(* Logix 5000 project; controller LeakTestAuto vendor 1 type 14 code 226 rev 37.11; software revision 37.01; part 10 of 13 *)
(* tags used below, declared in another part *)
   AOI_Barcode_Comms : AOI_CommStatus;
   AOI_CTS1 : AOI_CTS_INSTRUMENT;
   AOI_CTS1_Comms : AOI_CommStatus;
   AOI_CTS2 : AOI_CTS_INSTRUMENT;
   AOI_CTS2_Comms : AOI_CommStatus;
   AOI_RFID_Comms : AOI_CommStatus;
   AOI_Robot_Comms : AOI_CommStatus;
   AOI_SeqSteps : AOI_StandardSeqSteps;
   BarcodeScanner : udt_OutputStructure;
   Conveyor : udt_OutputStructure;
   Conveyor_Seq : udt_SequenceStructure_X64;
   ConveyorCleatSensorFault : BOOL;
   CTS1_Seq : udt_SequenceStructure_X64;
   CTS2_Seq : udt_SequenceStructure_X64;
   FailCount : COUNTER;
   LastFaults : DINT[2];
   LeakTester1 : udt_OutputStructure;
   LeakTester2 : udt_OutputStructure;
   Nest1Bypass : BOOL;
   Nest1Cylinder : udt_OutputStructure;
   Nest2Bypass : BOOL;
   Nest2Cylinder : udt_OutputStructure;
   ONS_ClearWarnings : BOOL;
   OP220 : udt_Mode;
   OP220_Fault_Counter : COUNTER;
   OP220_Fault_Counter_ONS : BOOL;
   OP220_Fault_Number : DINT;
   OP220_Fault_Reset_ONS : BOOL;
   OP220_FaultCounter_Reset_ONS : BOOL;
   OP220_HomingSeq : udt_SequenceStructure_X64;
   OP220_LeakTest : udt_ProcessFault;
   OP220_Seq : udt_SequenceStructure_X64;
   RFID_Cylinder1_Mismatch : BOOL;
   RFID_Cylinder2_Mismatch : BOOL;
   RFIDScanner : udt_OutputStructure;
   Robot : udt_OutputStructure;
   RobotGripper : udt_OutputStructure;
   TON_Cylinder1DownTimeout : TIMER;
   TON_Cylinder1UpTimeout : TIMER;
   TON_Cylinder2DownTimeout : TIMER;
   TON_Cylinder2UpTimeout : TIMER;
   TON_FailChute : TIMER[10];
   I_OP220_N3_REJECT_BIN_OK : ALIAS FOR Local:3:I.Pt09.Data;
   I_OP220_N4_DC_OK : ALIAS FOR Local:4:I.Pt01.Data;
   I_OP220_N4_DC_OK_PS2 : ALIAS FOR Local:4:I.Pt04.Data;
   OP220_ConsumedFromMain_RobotPickupSafe : BOOL;
   OP220_EStopTest_DCS : DCI_STOP;
   PLC : AOI_PLC;
   ShiftChange : BOOL;
(* MainProgram, continued *)

ROUTINE R90_Faults   (* ladder *)
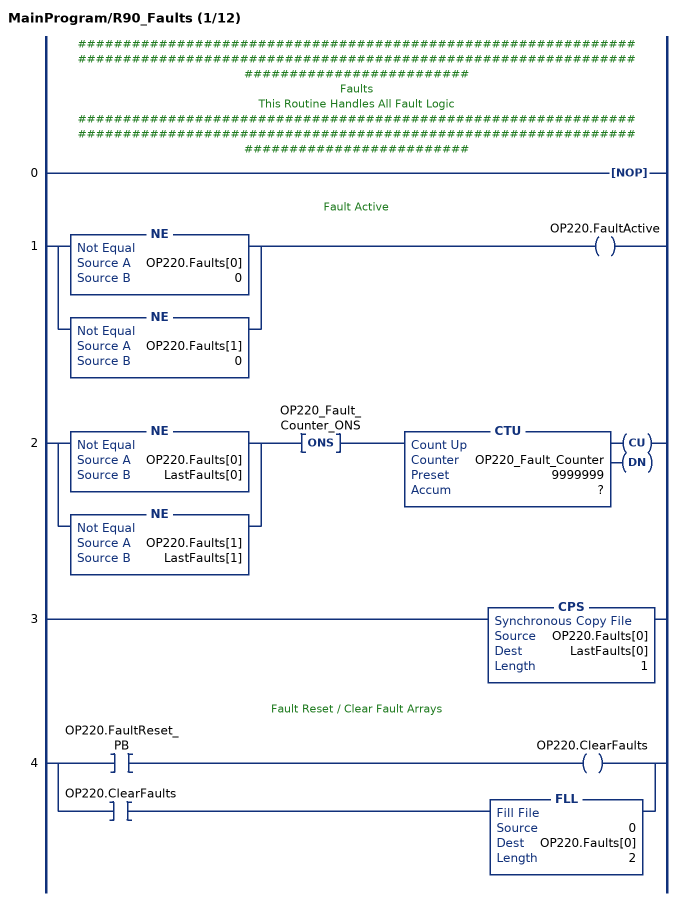
   // #####################################################################################################################################################
   // Faults
   // This Routine Handles All Fault Logic
   // #####################################################################################################################################################
   0: NOP();
   // Fault Active
   1: [NE(OP220.Faults[0],0) ,NE(OP220.Faults[1],0) ]OTE(OP220.FaultActive);
   2: [NE(OP220.Faults[0],LastFaults[0]) ,NE(OP220.Faults[1],LastFaults[1]) ]ONS(OP220_Fault_Counter_ONS)CTU(OP220_Fault_Counter,?,?);
   3: CPS(OP220.Faults[0],LastFaults[0],1);
   // Fault Reset / Clear Fault Arrays
   4: [XIC(OP220.FaultReset_PB) OTE(OP220.ClearFaults) ,XIC(OP220.ClearFaults) FLL(0,OP220.Faults[0],2) ];
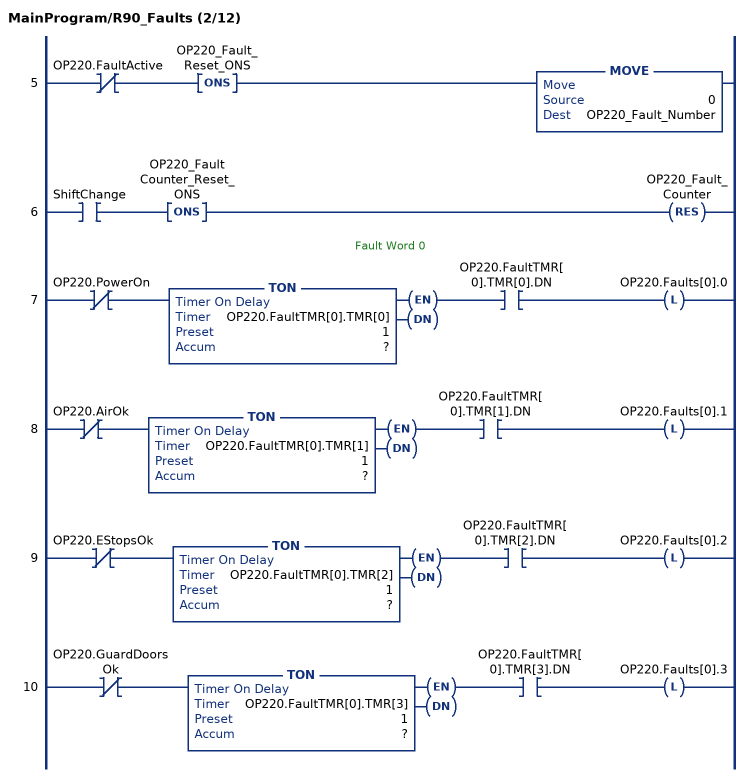
   5: XIO(OP220.FaultActive)ONS(OP220_Fault_Reset_ONS)MOVE(0,OP220_Fault_Number);
   6: XIC(ShiftChange)ONS(OP220_FaultCounter_Reset_ONS)RES(OP220_Fault_Counter);
   // Fault Word 0
   7: XIO(OP220.PowerOn)TON(OP220.FaultTMR[0].TMR[0],?,?)XIC(OP220.FaultTMR[0].TMR[0].DN)OTL(OP220.Faults[0].0);
   8: XIO(OP220.AirOk)TON(OP220.FaultTMR[0].TMR[1],?,?)XIC(OP220.FaultTMR[0].TMR[1].DN)OTL(OP220.Faults[0].1);
   9: XIO(OP220.EStopsOk)TON(OP220.FaultTMR[0].TMR[2],?,?)XIC(OP220.FaultTMR[0].TMR[2].DN)OTL(OP220.Faults[0].2);
   10: XIO(OP220.GuardDoorsOk)TON(OP220.FaultTMR[0].TMR[3],?,?)XIC(OP220.FaultTMR[0].TMR[3].DN)OTL(OP220.Faults[0].3);
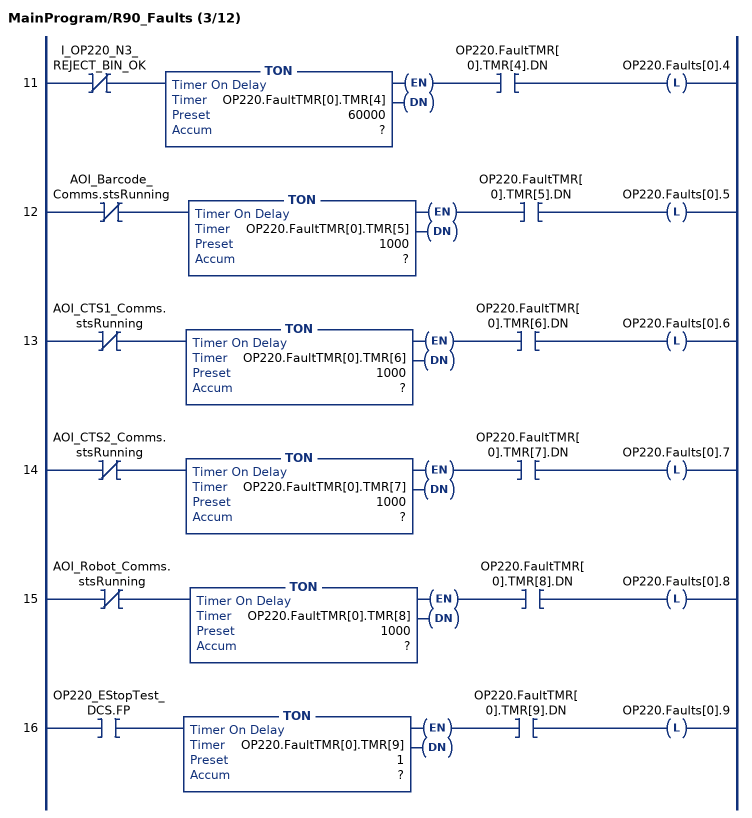
   11: XIO(I_OP220_N3_REJECT_BIN_OK)TON(OP220.FaultTMR[0].TMR[4],?,?)XIC(OP220.FaultTMR[0].TMR[4].DN)OTL(OP220.Faults[0].4);
   12: XIO(AOI_Barcode_Comms.stsRunning)TON(OP220.FaultTMR[0].TMR[5],?,?)XIC(OP220.FaultTMR[0].TMR[5].DN)OTL(OP220.Faults[0].5);
   13: XIO(AOI_CTS1_Comms.stsRunning)TON(OP220.FaultTMR[0].TMR[6],?,?)XIC(OP220.FaultTMR[0].TMR[6].DN)OTL(OP220.Faults[0].6);
   14: XIO(AOI_CTS2_Comms.stsRunning)TON(OP220.FaultTMR[0].TMR[7],?,?)XIC(OP220.FaultTMR[0].TMR[7].DN)OTL(OP220.Faults[0].7);
   15: XIO(AOI_Robot_Comms.stsRunning)TON(OP220.FaultTMR[0].TMR[8],?,?)XIC(OP220.FaultTMR[0].TMR[8].DN)OTL(OP220.Faults[0].8);
   16: XIC(OP220_EStopTest_DCS.FP)TON(OP220.FaultTMR[0].TMR[9],?,?)XIC(OP220.FaultTMR[0].TMR[9].DN)OTL(OP220.Faults[0].9);
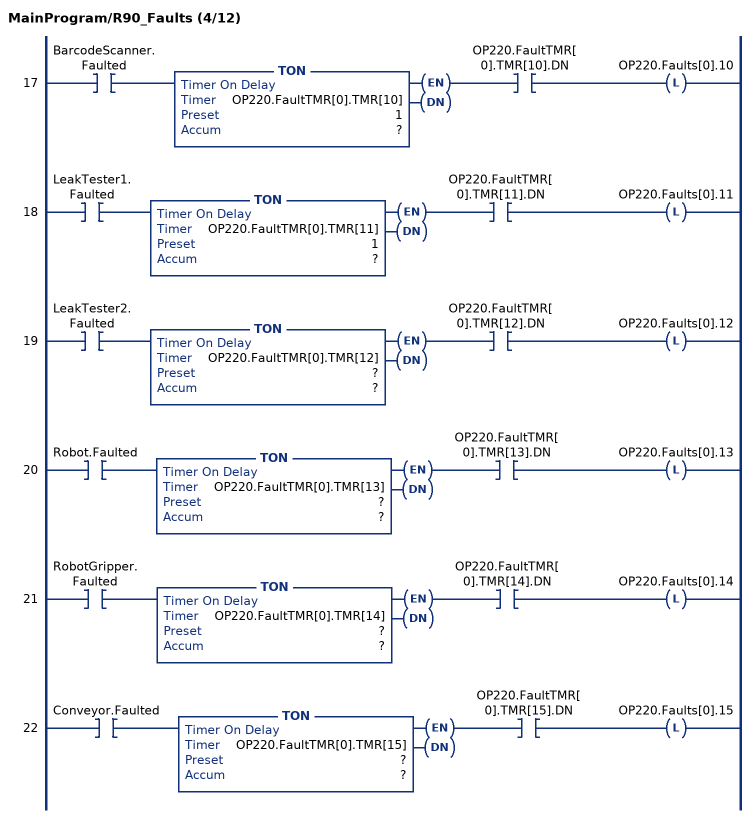
   17: XIC(BarcodeScanner.Faulted)TON(OP220.FaultTMR[0].TMR[10],?,?)XIC(OP220.FaultTMR[0].TMR[10].DN)OTL(OP220.Faults[0].10);
   18: XIC(LeakTester1.Faulted)TON(OP220.FaultTMR[0].TMR[11],?,?)XIC(OP220.FaultTMR[0].TMR[11].DN)OTL(OP220.Faults[0].11);
   19: XIC(LeakTester2.Faulted)TON(OP220.FaultTMR[0].TMR[12],?,?)XIC(OP220.FaultTMR[0].TMR[12].DN)OTL(OP220.Faults[0].12);
   20: XIC(Robot.Faulted)TON(OP220.FaultTMR[0].TMR[13],?,?)XIC(OP220.FaultTMR[0].TMR[13].DN)OTL(OP220.Faults[0].13);
   21: XIC(RobotGripper.Faulted)TON(OP220.FaultTMR[0].TMR[14],?,?)XIC(OP220.FaultTMR[0].TMR[14].DN)OTL(OP220.Faults[0].14);
   22: XIC(Conveyor.Faulted)TON(OP220.FaultTMR[0].TMR[15],?,?)XIC(OP220.FaultTMR[0].TMR[15].DN)OTL(OP220.Faults[0].15);
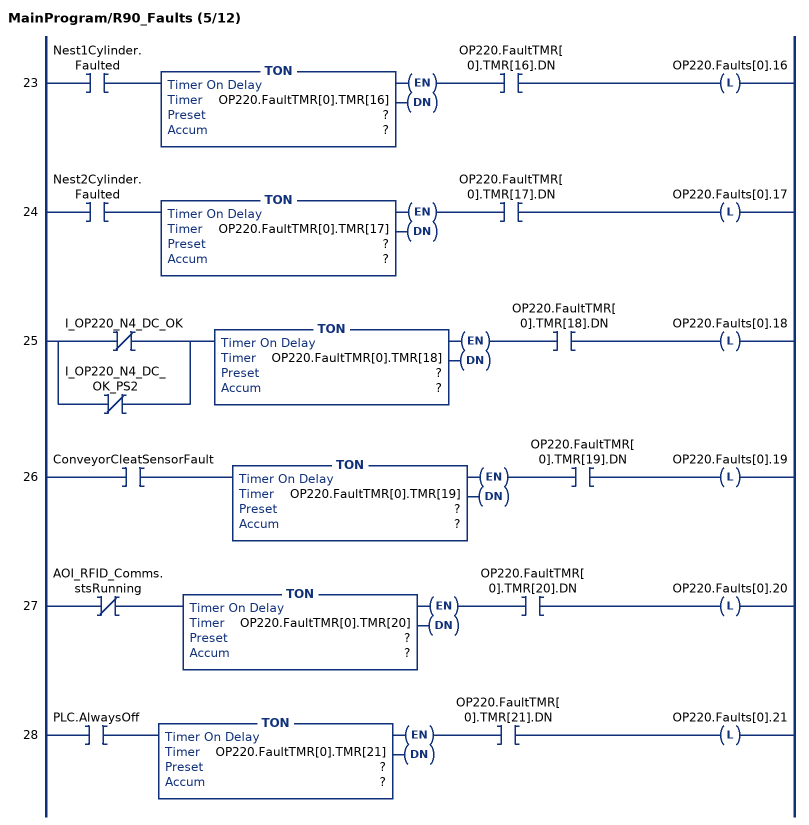
   23: XIC(Nest1Cylinder.Faulted)TON(OP220.FaultTMR[0].TMR[16],?,?)XIC(OP220.FaultTMR[0].TMR[16].DN)OTL(OP220.Faults[0].16);
   24: XIC(Nest2Cylinder.Faulted)TON(OP220.FaultTMR[0].TMR[17],?,?)XIC(OP220.FaultTMR[0].TMR[17].DN)OTL(OP220.Faults[0].17);
   25: [XIO(I_OP220_N4_DC_OK) ,XIO(I_OP220_N4_DC_OK_PS2) ]TON(OP220.FaultTMR[0].TMR[18],?,?)XIC(OP220.FaultTMR[0].TMR[18].DN)OTL(OP220.Faults[0].18);
   26: XIC(ConveyorCleatSensorFault)TON(OP220.FaultTMR[0].TMR[19],?,?)XIC(OP220.FaultTMR[0].TMR[19].DN)OTL(OP220.Faults[0].19);
   27: XIO(AOI_RFID_Comms.stsRunning)TON(OP220.FaultTMR[0].TMR[20],?,?)XIC(OP220.FaultTMR[0].TMR[20].DN)OTL(OP220.Faults[0].20);
   28: XIC(PLC.AlwaysOff)TON(OP220.FaultTMR[0].TMR[21],?,?)XIC(OP220.FaultTMR[0].TMR[21].DN)OTL(OP220.Faults[0].21);
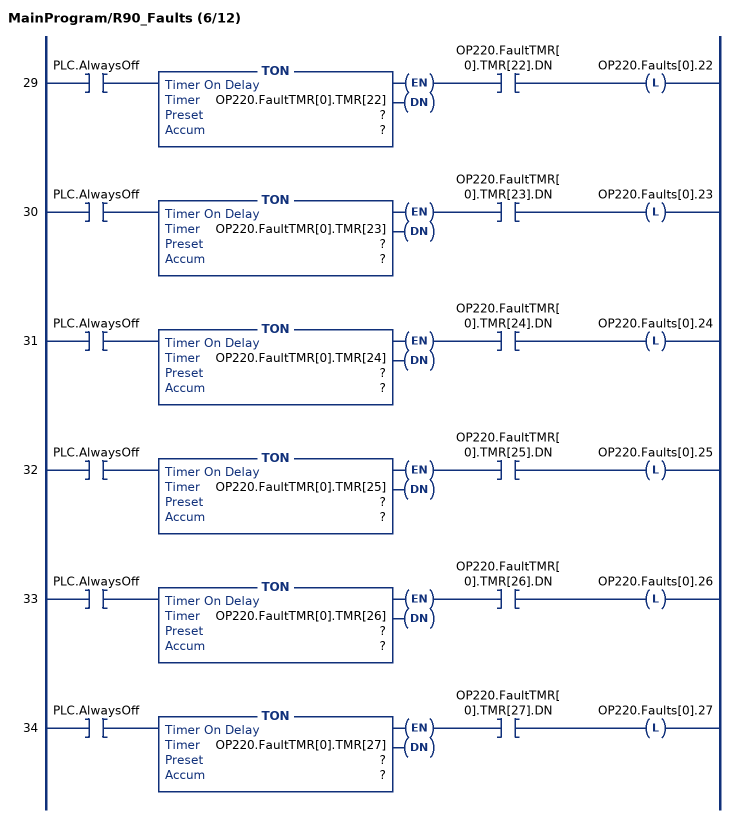
   29: XIC(PLC.AlwaysOff)TON(OP220.FaultTMR[0].TMR[22],?,?)XIC(OP220.FaultTMR[0].TMR[22].DN)OTL(OP220.Faults[0].22);
   30: XIC(PLC.AlwaysOff)TON(OP220.FaultTMR[0].TMR[23],?,?)XIC(OP220.FaultTMR[0].TMR[23].DN)OTL(OP220.Faults[0].23);
   31: XIC(PLC.AlwaysOff)TON(OP220.FaultTMR[0].TMR[24],?,?)XIC(OP220.FaultTMR[0].TMR[24].DN)OTL(OP220.Faults[0].24);
   32: XIC(PLC.AlwaysOff)TON(OP220.FaultTMR[0].TMR[25],?,?)XIC(OP220.FaultTMR[0].TMR[25].DN)OTL(OP220.Faults[0].25);
   33: XIC(PLC.AlwaysOff)TON(OP220.FaultTMR[0].TMR[26],?,?)XIC(OP220.FaultTMR[0].TMR[26].DN)OTL(OP220.Faults[0].26);
   34: XIC(PLC.AlwaysOff)TON(OP220.FaultTMR[0].TMR[27],?,?)XIC(OP220.FaultTMR[0].TMR[27].DN)OTL(OP220.Faults[0].27);
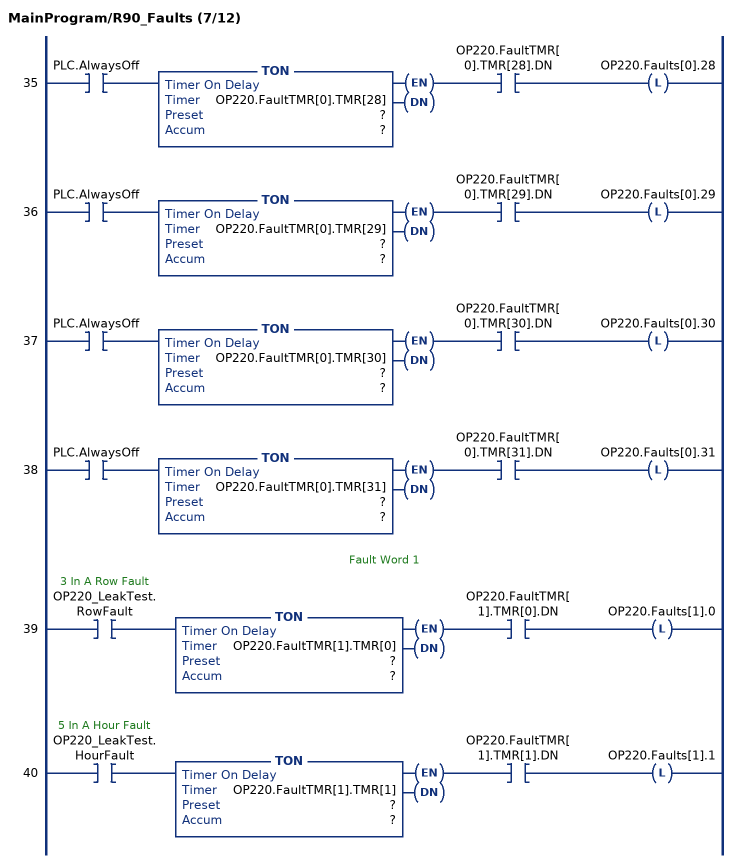
   35: XIC(PLC.AlwaysOff)TON(OP220.FaultTMR[0].TMR[28],?,?)XIC(OP220.FaultTMR[0].TMR[28].DN)OTL(OP220.Faults[0].28);
   36: XIC(PLC.AlwaysOff)TON(OP220.FaultTMR[0].TMR[29],?,?)XIC(OP220.FaultTMR[0].TMR[29].DN)OTL(OP220.Faults[0].29);
   37: XIC(PLC.AlwaysOff)TON(OP220.FaultTMR[0].TMR[30],?,?)XIC(OP220.FaultTMR[0].TMR[30].DN)OTL(OP220.Faults[0].30);
   38: XIC(PLC.AlwaysOff)TON(OP220.FaultTMR[0].TMR[31],?,?)XIC(OP220.FaultTMR[0].TMR[31].DN)OTL(OP220.Faults[0].31);
   // Fault Word 1
   39: XIC(OP220_LeakTest.RowFault)TON(OP220.FaultTMR[1].TMR[0],?,?)XIC(OP220.FaultTMR[1].TMR[0].DN)OTL(OP220.Faults[1].0);
   40: XIC(OP220_LeakTest.HourFault)TON(OP220.FaultTMR[1].TMR[1],?,?)XIC(OP220.FaultTMR[1].TMR[1].DN)OTL(OP220.Faults[1].1);
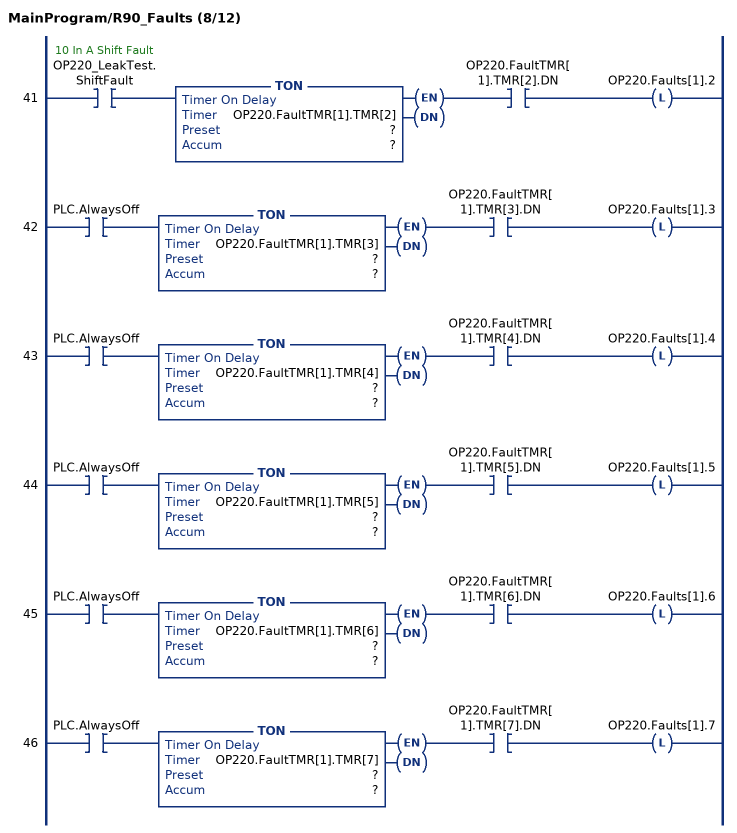
   41: XIC(OP220_LeakTest.ShiftFault)TON(OP220.FaultTMR[1].TMR[2],?,?)XIC(OP220.FaultTMR[1].TMR[2].DN)OTL(OP220.Faults[1].2);
   42: XIC(PLC.AlwaysOff)TON(OP220.FaultTMR[1].TMR[3],?,?)XIC(OP220.FaultTMR[1].TMR[3].DN)OTL(OP220.Faults[1].3);
   43: XIC(PLC.AlwaysOff)TON(OP220.FaultTMR[1].TMR[4],?,?)XIC(OP220.FaultTMR[1].TMR[4].DN)OTL(OP220.Faults[1].4);
   44: XIC(PLC.AlwaysOff)TON(OP220.FaultTMR[1].TMR[5],?,?)XIC(OP220.FaultTMR[1].TMR[5].DN)OTL(OP220.Faults[1].5);
   45: XIC(PLC.AlwaysOff)TON(OP220.FaultTMR[1].TMR[6],?,?)XIC(OP220.FaultTMR[1].TMR[6].DN)OTL(OP220.Faults[1].6);
   46: XIC(PLC.AlwaysOff)TON(OP220.FaultTMR[1].TMR[7],?,?)XIC(OP220.FaultTMR[1].TMR[7].DN)OTL(OP220.Faults[1].7);
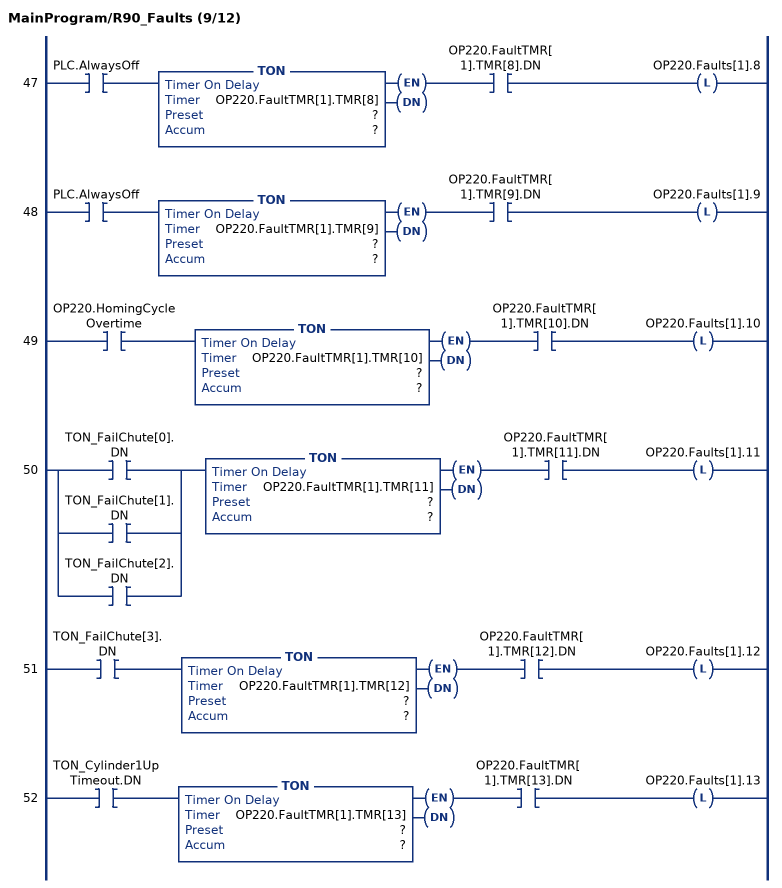
   47: XIC(PLC.AlwaysOff)TON(OP220.FaultTMR[1].TMR[8],?,?)XIC(OP220.FaultTMR[1].TMR[8].DN)OTL(OP220.Faults[1].8);
   48: XIC(PLC.AlwaysOff)TON(OP220.FaultTMR[1].TMR[9],?,?)XIC(OP220.FaultTMR[1].TMR[9].DN)OTL(OP220.Faults[1].9);
   49: XIC(OP220.HomingCycleOvertime)TON(OP220.FaultTMR[1].TMR[10],?,?)XIC(OP220.FaultTMR[1].TMR[10].DN)OTL(OP220.Faults[1].10);
   50: [XIC(TON_FailChute[0].DN) ,XIC(TON_FailChute[1].DN) ,XIC(TON_FailChute[2].DN) ]TON(OP220.FaultTMR[1].TMR[11],?,?)XIC(OP220.FaultTMR[1].TMR[11].DN)OTL(OP220.Faults[1].11);
   51: XIC(TON_FailChute[3].DN)TON(OP220.FaultTMR[1].TMR[12],?,?)XIC(OP220.FaultTMR[1].TMR[12].DN)OTL(OP220.Faults[1].12);
   52: XIC(TON_Cylinder1UpTimeout.DN)TON(OP220.FaultTMR[1].TMR[13],?,?)XIC(OP220.FaultTMR[1].TMR[13].DN)OTL(OP220.Faults[1].13);
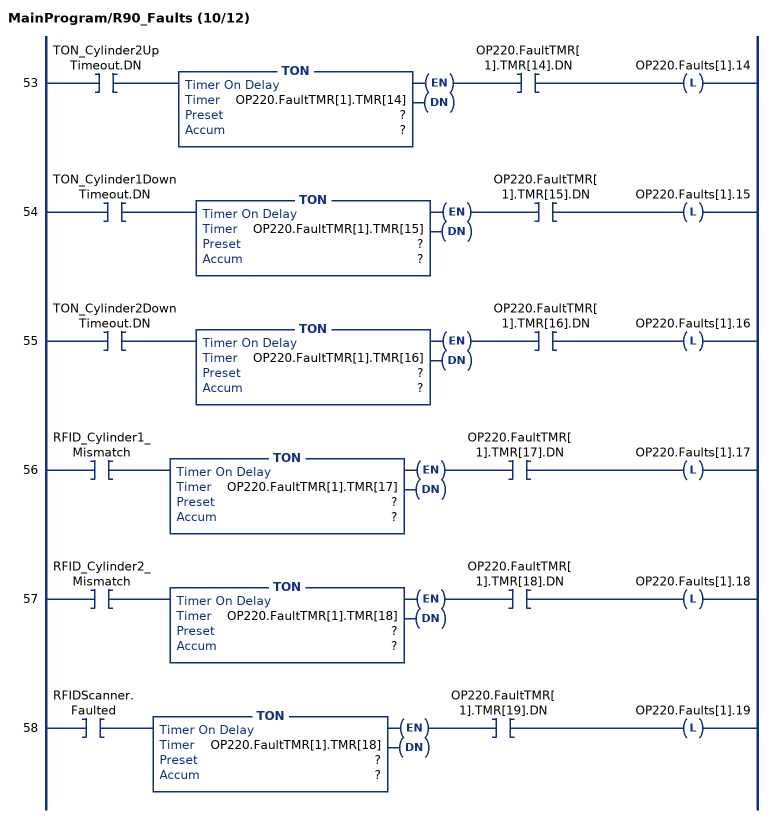
   53: XIC(TON_Cylinder2UpTimeout.DN)TON(OP220.FaultTMR[1].TMR[14],?,?)XIC(OP220.FaultTMR[1].TMR[14].DN)OTL(OP220.Faults[1].14);
   54: XIC(TON_Cylinder1DownTimeout.DN)TON(OP220.FaultTMR[1].TMR[15],?,?)XIC(OP220.FaultTMR[1].TMR[15].DN)OTL(OP220.Faults[1].15);
   55: XIC(TON_Cylinder2DownTimeout.DN)TON(OP220.FaultTMR[1].TMR[16],?,?)XIC(OP220.FaultTMR[1].TMR[16].DN)OTL(OP220.Faults[1].16);
   56: XIC(RFID_Cylinder1_Mismatch)TON(OP220.FaultTMR[1].TMR[17],?,?)XIC(OP220.FaultTMR[1].TMR[17].DN)OTL(OP220.Faults[1].17);
   57: XIC(RFID_Cylinder2_Mismatch)TON(OP220.FaultTMR[1].TMR[18],?,?)XIC(OP220.FaultTMR[1].TMR[18].DN)OTL(OP220.Faults[1].18);
   58: XIC(RFIDScanner.Faulted)TON(OP220.FaultTMR[1].TMR[18],?,?)XIC(OP220.FaultTMR[1].TMR[19].DN)OTL(OP220.Faults[1].19);
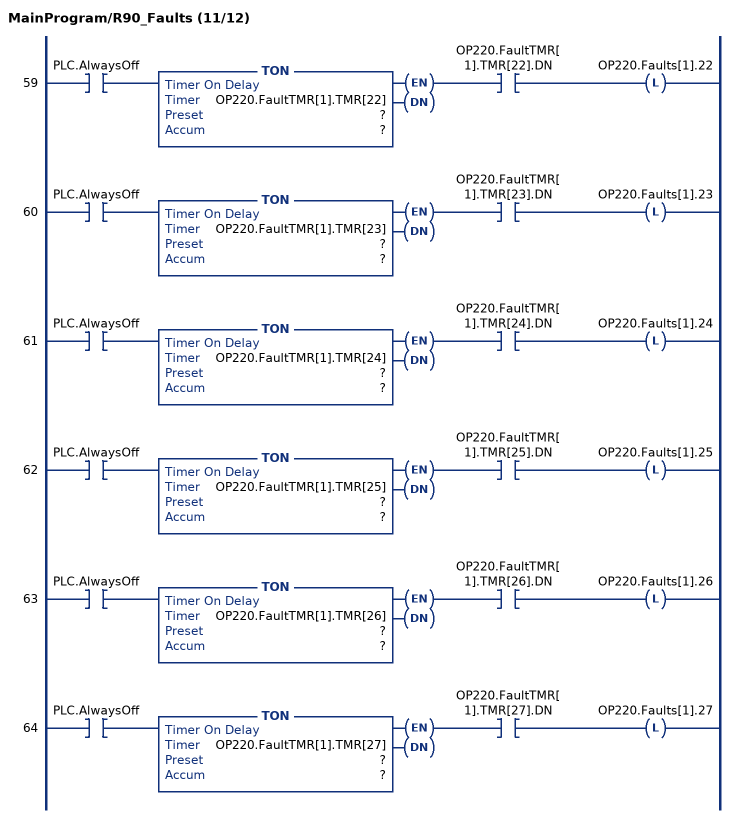
   59: XIC(PLC.AlwaysOff)TON(OP220.FaultTMR[1].TMR[22],?,?)XIC(OP220.FaultTMR[1].TMR[22].DN)OTL(OP220.Faults[1].22);
   60: XIC(PLC.AlwaysOff)TON(OP220.FaultTMR[1].TMR[23],?,?)XIC(OP220.FaultTMR[1].TMR[23].DN)OTL(OP220.Faults[1].23);
   61: XIC(PLC.AlwaysOff)TON(OP220.FaultTMR[1].TMR[24],?,?)XIC(OP220.FaultTMR[1].TMR[24].DN)OTL(OP220.Faults[1].24);
   62: XIC(PLC.AlwaysOff)TON(OP220.FaultTMR[1].TMR[25],?,?)XIC(OP220.FaultTMR[1].TMR[25].DN)OTL(OP220.Faults[1].25);
   63: XIC(PLC.AlwaysOff)TON(OP220.FaultTMR[1].TMR[26],?,?)XIC(OP220.FaultTMR[1].TMR[26].DN)OTL(OP220.Faults[1].26);
   64: XIC(PLC.AlwaysOff)TON(OP220.FaultTMR[1].TMR[27],?,?)XIC(OP220.FaultTMR[1].TMR[27].DN)OTL(OP220.Faults[1].27);
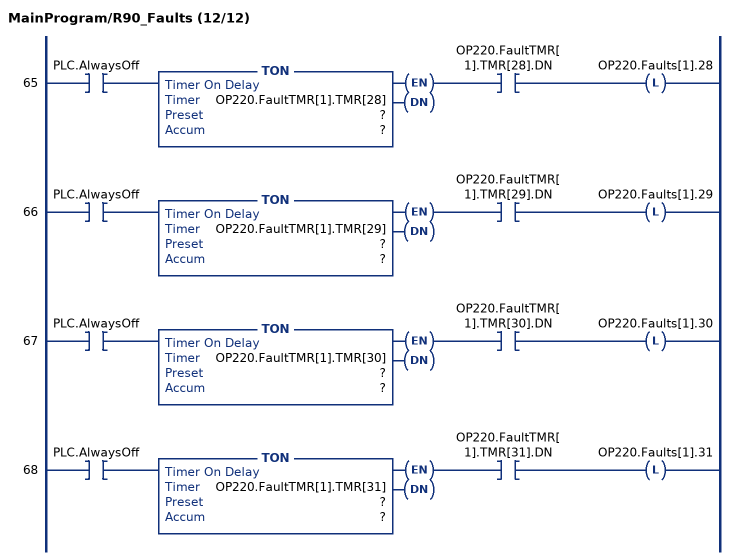
   65: XIC(PLC.AlwaysOff)TON(OP220.FaultTMR[1].TMR[28],?,?)XIC(OP220.FaultTMR[1].TMR[28].DN)OTL(OP220.Faults[1].28);
   66: XIC(PLC.AlwaysOff)TON(OP220.FaultTMR[1].TMR[29],?,?)XIC(OP220.FaultTMR[1].TMR[29].DN)OTL(OP220.Faults[1].29);
   67: XIC(PLC.AlwaysOff)TON(OP220.FaultTMR[1].TMR[30],?,?)XIC(OP220.FaultTMR[1].TMR[30].DN)OTL(OP220.Faults[1].30);
   68: XIC(PLC.AlwaysOff)TON(OP220.FaultTMR[1].TMR[31],?,?)XIC(OP220.FaultTMR[1].TMR[31].DN)OTL(OP220.Faults[1].31);
END_ROUTINE

ROUTINE R91_Warnings   (* ladder *)
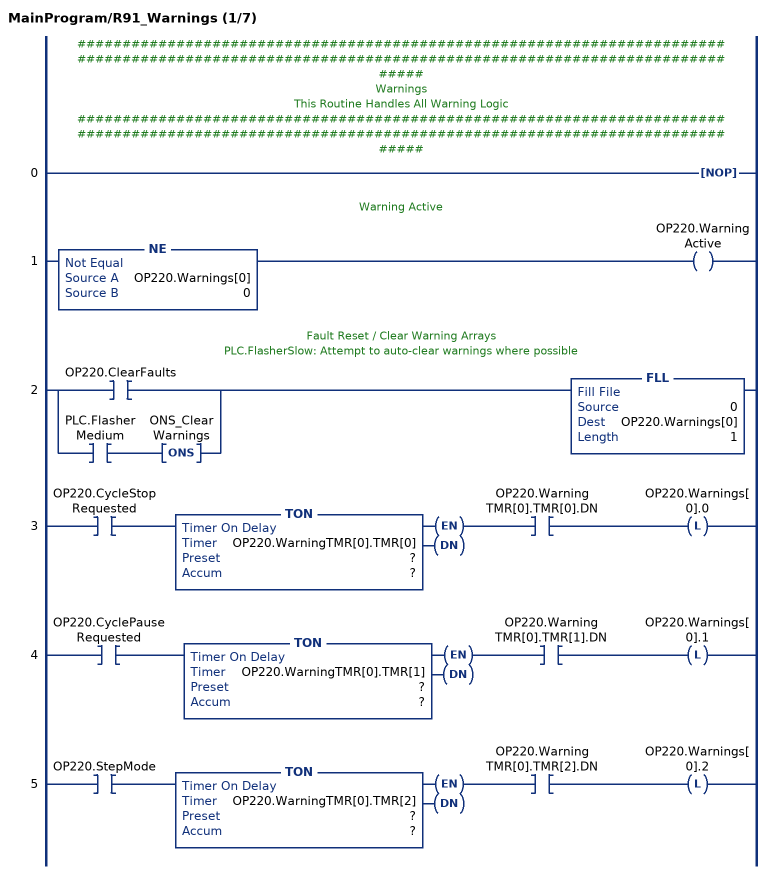
   // #####################################################################################################################################################
   // Warnings
   // This Routine Handles All Warning Logic
   // #####################################################################################################################################################
   0: NOP();
   // Warning Active
   1: NE(OP220.Warnings[0],0)OTE(OP220.WarningActive);
   // Fault Reset / Clear Warning Arrays
   // PLC.FlasherSlow: Attempt to auto-clear warnings where possible
   2: [XIC(OP220.ClearFaults) ,XIC(PLC.FlasherMedium) ONS(ONS_ClearWarnings) ]FLL(0,OP220.Warnings[0],1);
   3: XIC(OP220.CycleStopRequested)TON(OP220.WarningTMR[0].TMR[0],?,?)XIC(OP220.WarningTMR[0].TMR[0].DN)OTL(OP220.Warnings[0].0);
   4: XIC(OP220.CyclePauseRequested)TON(OP220.WarningTMR[0].TMR[1],?,?)XIC(OP220.WarningTMR[0].TMR[1].DN)OTL(OP220.Warnings[0].1);
   5: XIC(OP220.StepMode)TON(OP220.WarningTMR[0].TMR[2],?,?)XIC(OP220.WarningTMR[0].TMR[2].DN)OTL(OP220.Warnings[0].2);
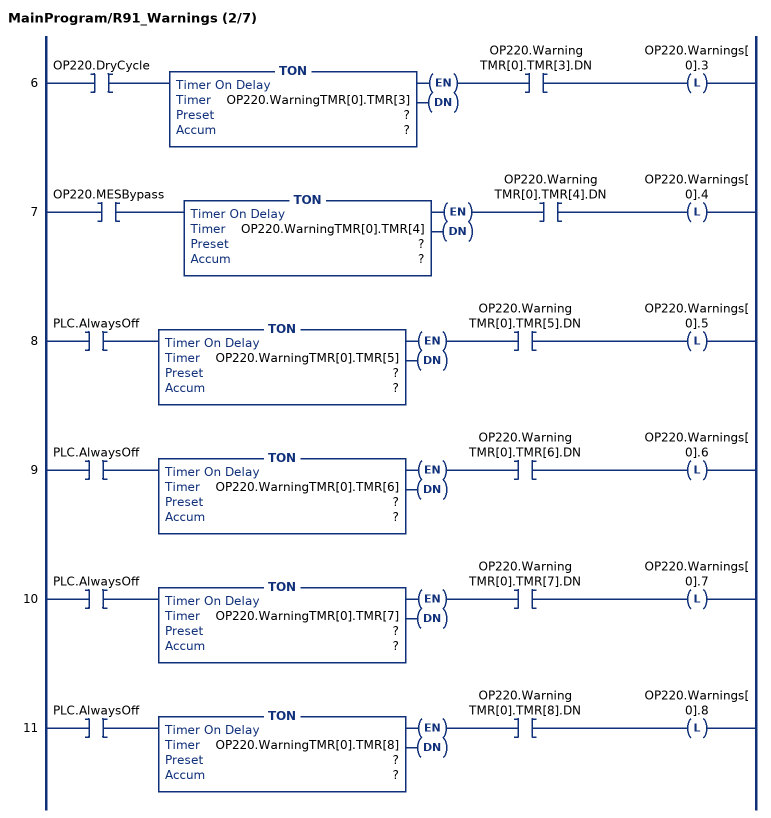
   6: XIC(OP220.DryCycle)TON(OP220.WarningTMR[0].TMR[3],?,?)XIC(OP220.WarningTMR[0].TMR[3].DN)OTL(OP220.Warnings[0].3);
   7: XIC(OP220.MESBypass)TON(OP220.WarningTMR[0].TMR[4],?,?)XIC(OP220.WarningTMR[0].TMR[4].DN)OTL(OP220.Warnings[0].4);
   8: XIC(PLC.AlwaysOff)TON(OP220.WarningTMR[0].TMR[5],?,?)XIC(OP220.WarningTMR[0].TMR[5].DN)OTL(OP220.Warnings[0].5);
   9: XIC(PLC.AlwaysOff)TON(OP220.WarningTMR[0].TMR[6],?,?)XIC(OP220.WarningTMR[0].TMR[6].DN)OTL(OP220.Warnings[0].6);
   10: XIC(PLC.AlwaysOff)TON(OP220.WarningTMR[0].TMR[7],?,?)XIC(OP220.WarningTMR[0].TMR[7].DN)OTL(OP220.Warnings[0].7);
   11: XIC(PLC.AlwaysOff)TON(OP220.WarningTMR[0].TMR[8],?,?)XIC(OP220.WarningTMR[0].TMR[8].DN)OTL(OP220.Warnings[0].8);
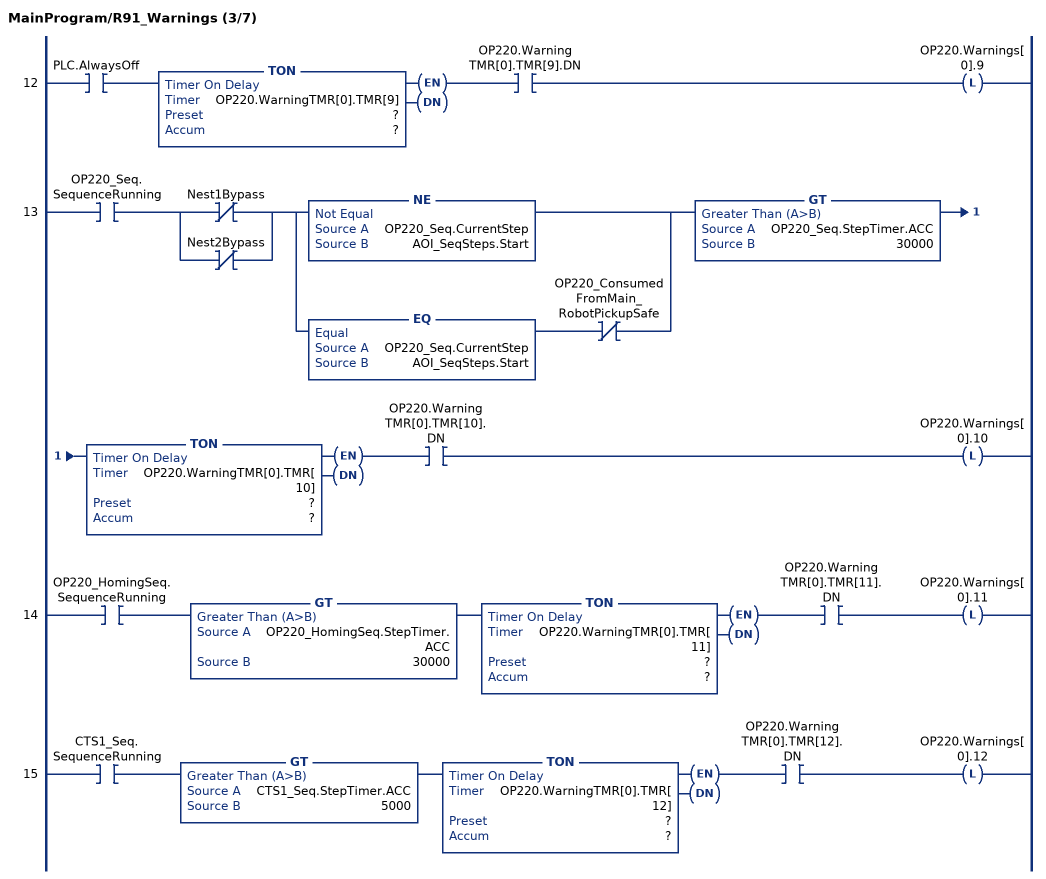
   12: XIC(PLC.AlwaysOff)TON(OP220.WarningTMR[0].TMR[9],?,?)XIC(OP220.WarningTMR[0].TMR[9].DN)OTL(OP220.Warnings[0].9);
   13: XIC(OP220_Seq.SequenceRunning)[XIO(Nest1Bypass) ,XIO(Nest2Bypass) ][NE(OP220_Seq.CurrentStep,AOI_SeqSteps.Start) ,EQ(OP220_Seq.CurrentStep,AOI_SeqSteps.Start) XIO(OP220_ConsumedFromMain_RobotPickupSafe) ]GT(OP220_Seq.StepTimer.ACC,30000)TON(OP220.WarningTMR[0].TMR[10],?,?)XIC(OP220.WarningTMR[0].TMR[10].DN)OTL(OP220.Warnings[0].10);
   14: XIC(OP220_HomingSeq.SequenceRunning)GT(OP220_HomingSeq.StepTimer.ACC,30000)TON(OP220.WarningTMR[0].TMR[11],?,?)XIC(OP220.WarningTMR[0].TMR[11].DN)OTL(OP220.Warnings[0].11);
   15: XIC(CTS1_Seq.SequenceRunning)GT(CTS1_Seq.StepTimer.ACC,5000)TON(OP220.WarningTMR[0].TMR[12],?,?)XIC(OP220.WarningTMR[0].TMR[12].DN)OTL(OP220.Warnings[0].12);
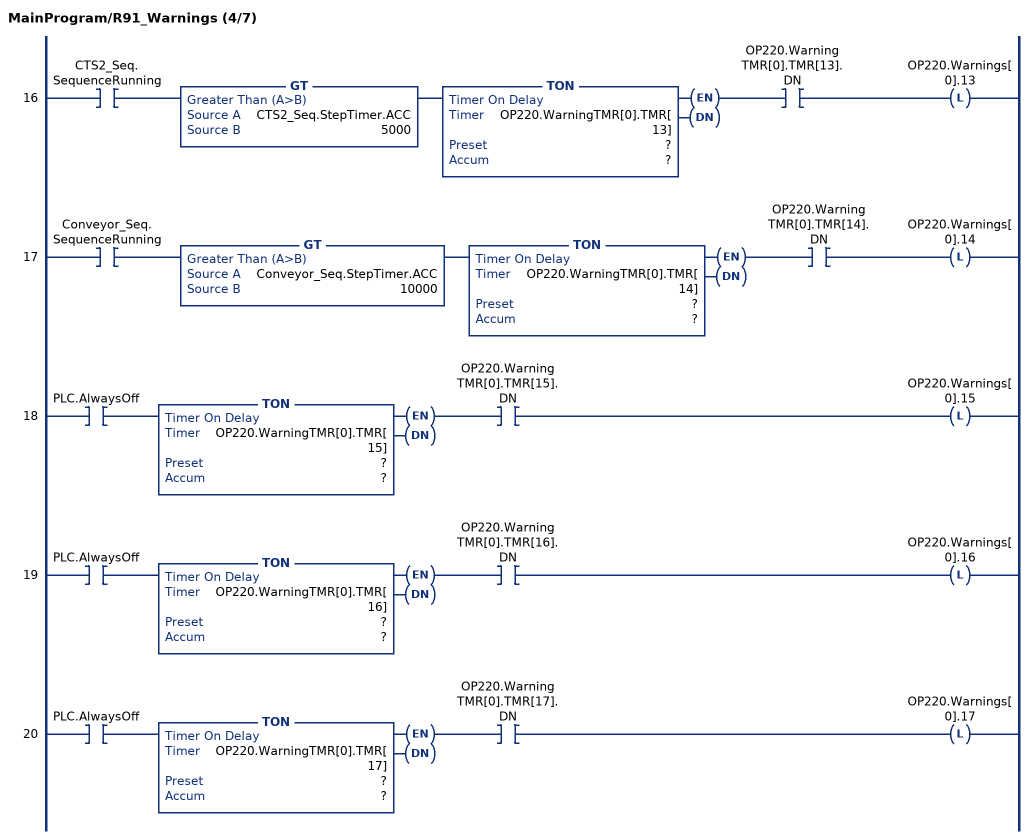
   16: XIC(CTS2_Seq.SequenceRunning)GT(CTS2_Seq.StepTimer.ACC,5000)TON(OP220.WarningTMR[0].TMR[13],?,?)XIC(OP220.WarningTMR[0].TMR[13].DN)OTL(OP220.Warnings[0].13);
   17: XIC(Conveyor_Seq.SequenceRunning)GT(Conveyor_Seq.StepTimer.ACC,10000)TON(OP220.WarningTMR[0].TMR[14],?,?)XIC(OP220.WarningTMR[0].TMR[14].DN)OTL(OP220.Warnings[0].14);
   18: XIC(PLC.AlwaysOff)TON(OP220.WarningTMR[0].TMR[15],?,?)XIC(OP220.WarningTMR[0].TMR[15].DN)OTL(OP220.Warnings[0].15);
   19: XIC(PLC.AlwaysOff)TON(OP220.WarningTMR[0].TMR[16],?,?)XIC(OP220.WarningTMR[0].TMR[16].DN)OTL(OP220.Warnings[0].16);
   20: XIC(PLC.AlwaysOff)TON(OP220.WarningTMR[0].TMR[17],?,?)XIC(OP220.WarningTMR[0].TMR[17].DN)OTL(OP220.Warnings[0].17);
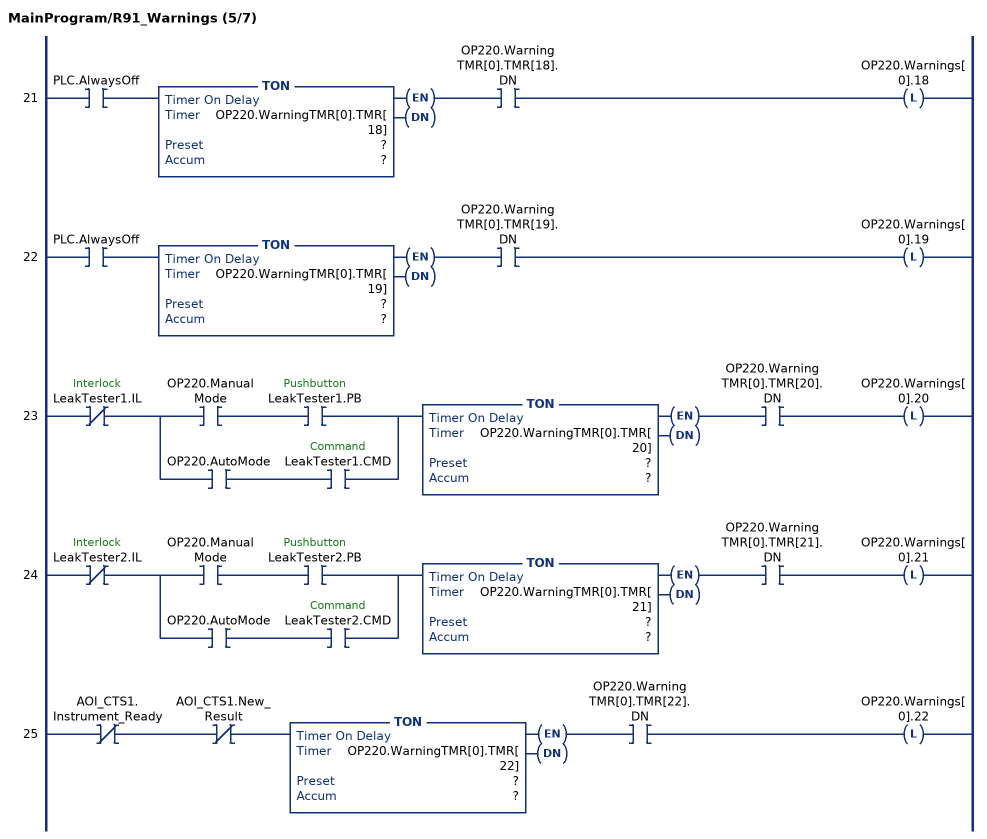
   21: XIC(PLC.AlwaysOff)TON(OP220.WarningTMR[0].TMR[18],?,?)XIC(OP220.WarningTMR[0].TMR[18].DN)OTL(OP220.Warnings[0].18);
   22: XIC(PLC.AlwaysOff)TON(OP220.WarningTMR[0].TMR[19],?,?)XIC(OP220.WarningTMR[0].TMR[19].DN)OTL(OP220.Warnings[0].19);
   23: XIO(LeakTester1.IL)[XIC(OP220.ManualMode) XIC(LeakTester1.PB) ,XIC(OP220.AutoMode) XIC(LeakTester1.CMD) ]TON(OP220.WarningTMR[0].TMR[20],?,?)XIC(OP220.WarningTMR[0].TMR[20].DN)OTL(OP220.Warnings[0].20);
   24: XIO(LeakTester2.IL)[XIC(OP220.ManualMode) XIC(LeakTester2.PB) ,XIC(OP220.AutoMode) XIC(LeakTester2.CMD) ]TON(OP220.WarningTMR[0].TMR[21],?,?)XIC(OP220.WarningTMR[0].TMR[21].DN)OTL(OP220.Warnings[0].21);
   25: XIO(AOI_CTS1.Instrument_Ready)XIO(AOI_CTS1.New_Result)TON(OP220.WarningTMR[0].TMR[22],?,?)XIC(OP220.WarningTMR[0].TMR[22].DN)OTL(OP220.Warnings[0].22);
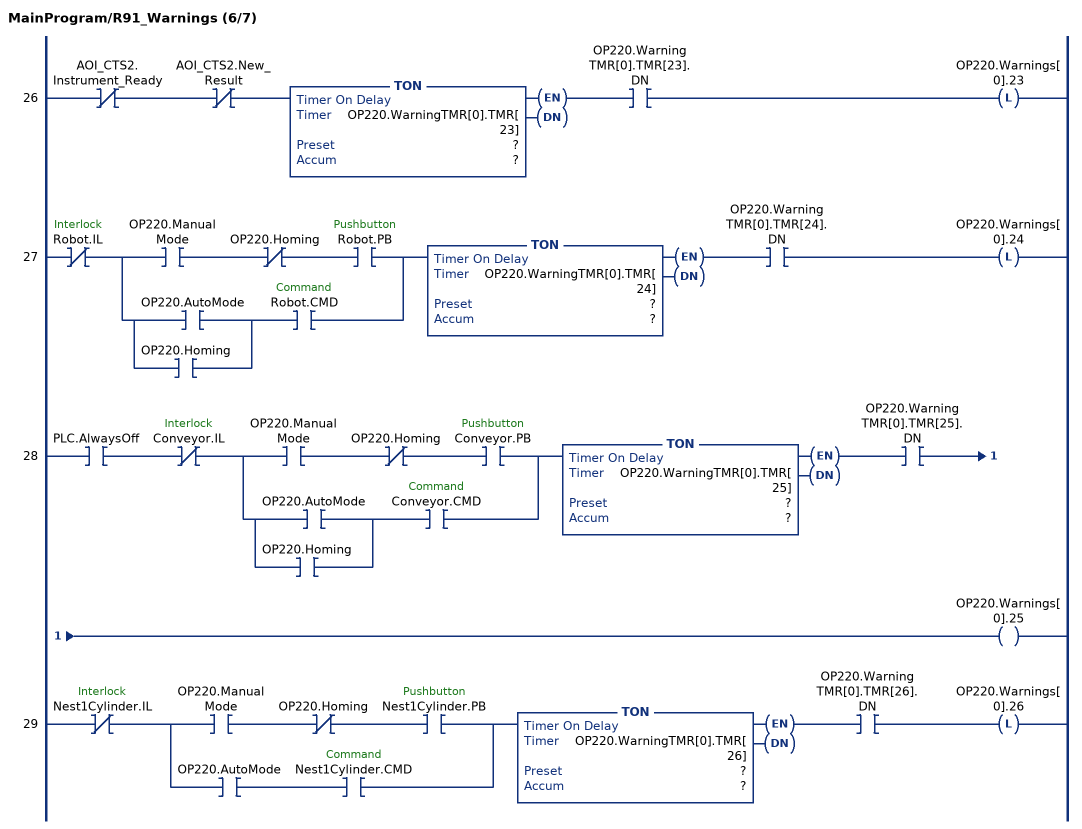
   26: XIO(AOI_CTS2.Instrument_Ready)XIO(AOI_CTS2.New_Result)TON(OP220.WarningTMR[0].TMR[23],?,?)XIC(OP220.WarningTMR[0].TMR[23].DN)OTL(OP220.Warnings[0].23);
   27: XIO(Robot.IL)[XIC(OP220.ManualMode) XIO(OP220.Homing) XIC(Robot.PB) ,[XIC(OP220.AutoMode) ,XIC(OP220.Homing) ] XIC(Robot.CMD) ]TON(OP220.WarningTMR[0].TMR[24],?,?)XIC(OP220.WarningTMR[0].TMR[24].DN)OTL(OP220.Warnings[0].24);
   28: XIC(PLC.AlwaysOff)XIO(Conveyor.IL)[XIC(OP220.ManualMode) XIO(OP220.Homing) XIC(Conveyor.PB) ,[XIC(OP220.AutoMode) ,XIC(OP220.Homing) ] XIC(Conveyor.CMD) ]TON(OP220.WarningTMR[0].TMR[25],?,?)XIC(OP220.WarningTMR[0].TMR[25].DN)OTE(OP220.Warnings[0].25);
   29: XIO(Nest1Cylinder.IL)[XIC(OP220.ManualMode) XIO(OP220.Homing) XIC(Nest1Cylinder.PB) ,XIC(OP220.AutoMode) XIC(Nest1Cylinder.CMD) ]TON(OP220.WarningTMR[0].TMR[26],?,?)XIC(OP220.WarningTMR[0].TMR[26].DN)OTL(OP220.Warnings[0].26);
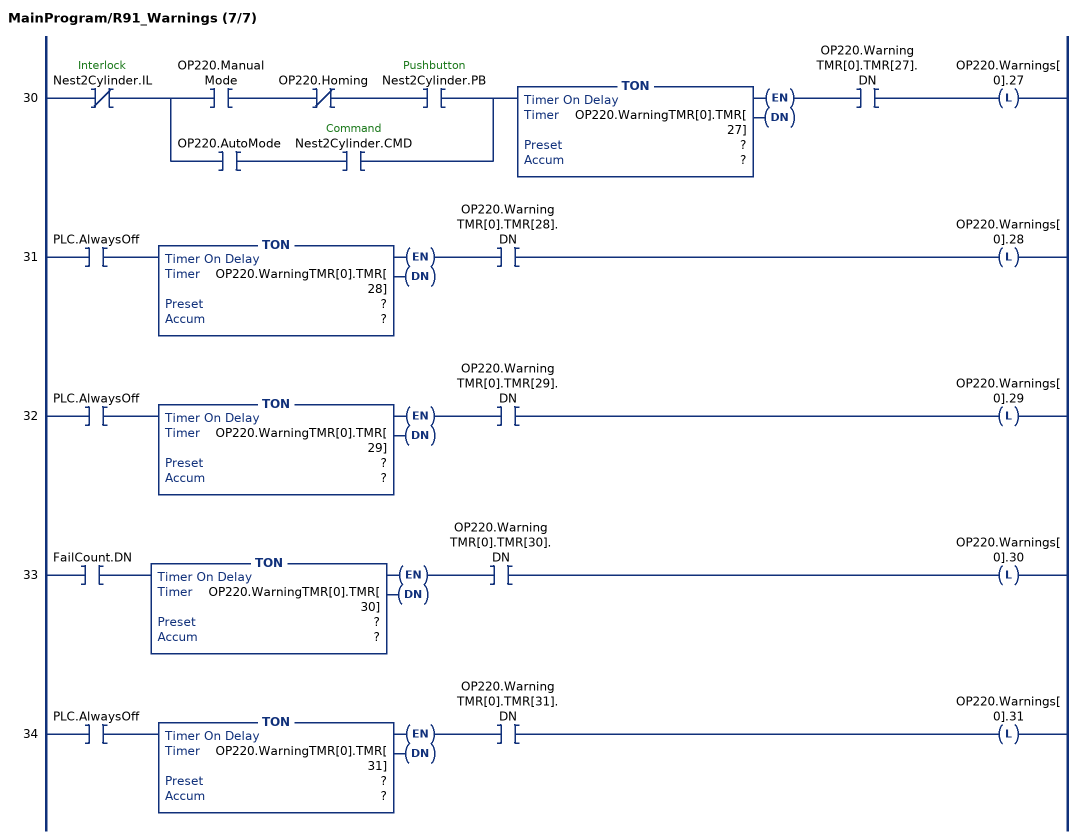
   30: XIO(Nest2Cylinder.IL)[XIC(OP220.ManualMode) XIO(OP220.Homing) XIC(Nest2Cylinder.PB) ,XIC(OP220.AutoMode) XIC(Nest2Cylinder.CMD) ]TON(OP220.WarningTMR[0].TMR[27],?,?)XIC(OP220.WarningTMR[0].TMR[27].DN)OTL(OP220.Warnings[0].27);
   31: XIC(PLC.AlwaysOff)TON(OP220.WarningTMR[0].TMR[28],?,?)XIC(OP220.WarningTMR[0].TMR[28].DN)OTL(OP220.Warnings[0].28);
   32: XIC(PLC.AlwaysOff)TON(OP220.WarningTMR[0].TMR[29],?,?)XIC(OP220.WarningTMR[0].TMR[29].DN)OTL(OP220.Warnings[0].29);
   33: XIC(FailCount.DN)TON(OP220.WarningTMR[0].TMR[30],?,?)XIC(OP220.WarningTMR[0].TMR[30].DN)OTL(OP220.Warnings[0].30);
   34: XIC(PLC.AlwaysOff)TON(OP220.WarningTMR[0].TMR[31],?,?)XIC(OP220.WarningTMR[0].TMR[31].DN)OTL(OP220.Warnings[0].31);
END_ROUTINE
